// SIMATIC S7-200 project (STEP 7-Micro/WIN), CPU 221 REL 01.10

SYMBOL_TABLE USER1
run              Q0.0
dir              Q0.1
s1               M5.0
s2               M5.1
s3               M5.2
p1               I0.0
p2               I0.1
p3               I0.2
END_SYMBOL_TABLE

ORGANIZATION_BLOCK MAIN:OB1
TITLE=PROGRAM COMMENTS
BEGIN
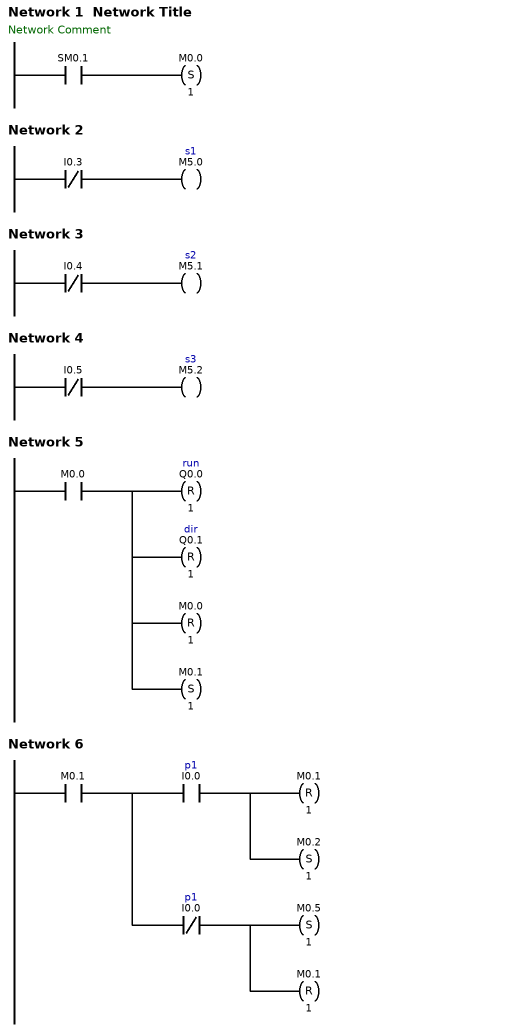
Network 1 // Network Title
// Network Comment
LD     SM0.1
S      M0.0, 1
Network 2
LDN    I0.3
=      s1:M5.0
Network 3
LDN    I0.4
=      s2:M5.1
Network 4
LDN    I0.5
=      s3:M5.2
Network 5
LD     M0.0
R      run:Q0.0, 1
R      dir:Q0.1, 1
R      M0.0, 1
S      M0.1, 1
Network 6
LD     M0.1
LPS
A      p1:I0.0
R      M0.1, 1
S      M0.2, 1
LPP
AN     p1:I0.0
S      M0.5, 1
R      M0.1, 1
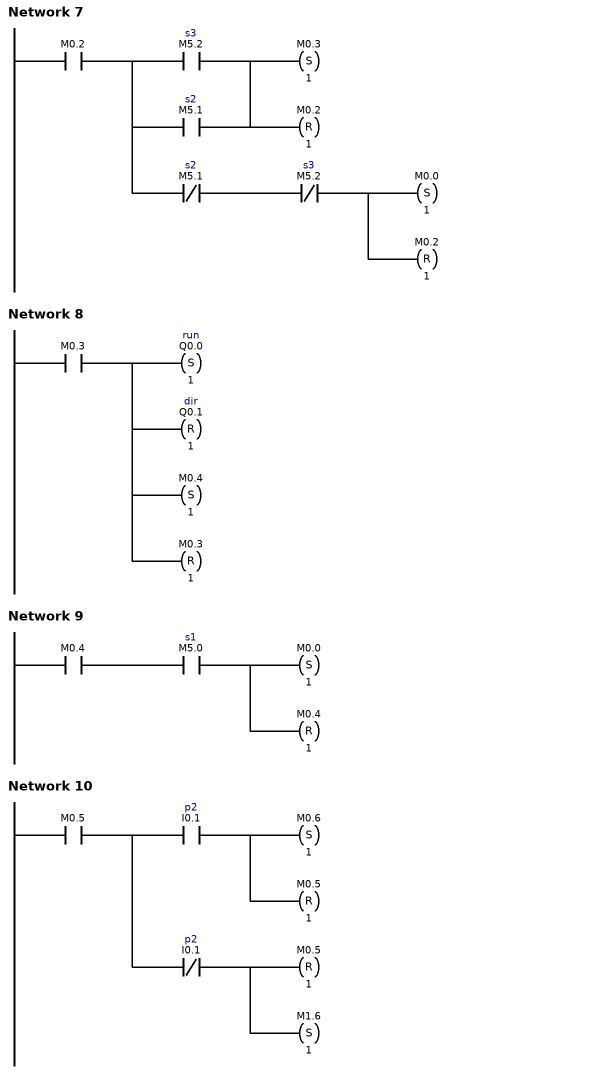
Network 7
LD     M0.2
LPS
LD     s3:M5.2
O      s2:M5.1
ALD
S      M0.3, 1
R      M0.2, 1
LPP
AN     s2:M5.1
AN     s3:M5.2
S      M0.0, 1
R      M0.2, 1
Network 8
LD     M0.3
S      run:Q0.0, 1
R      dir:Q0.1, 1
S      M0.4, 1
R      M0.3, 1
Network 9
LD     M0.4
A      s1:M5.0
S      M0.0, 1
R      M0.4, 1
Network 10
LD     M0.5
LPS
A      p2:I0.1
S      M0.6, 1
R      M0.5, 1
LPP
AN     p2:I0.1
R      M0.5, 1
S      M1.6, 1
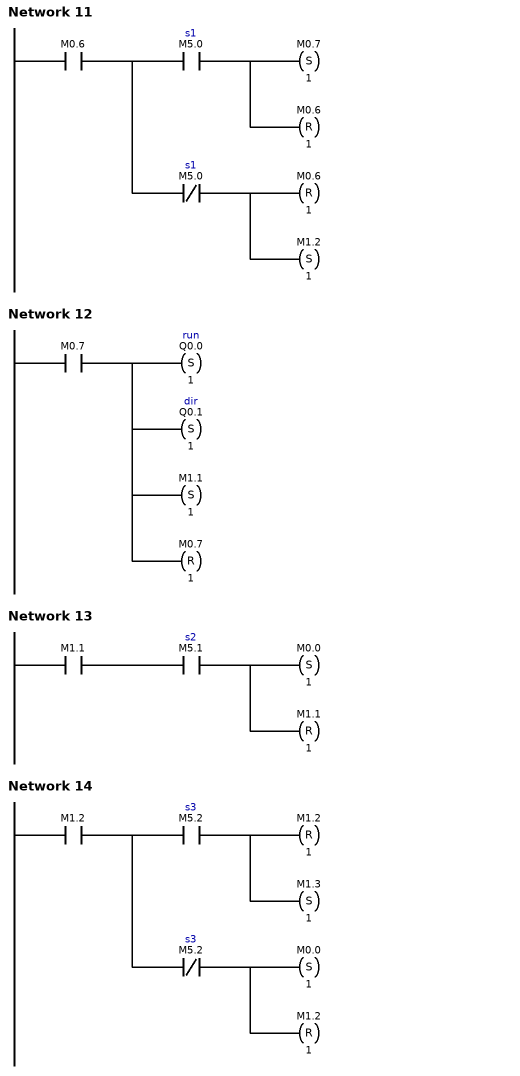
Network 11
LD     M0.6
LPS
A      s1:M5.0
S      M0.7, 1
R      M0.6, 1
LPP
AN     s1:M5.0
R      M0.6, 1
S      M1.2, 1
Network 12
LD     M0.7
S      run:Q0.0, 1
S      dir:Q0.1, 1
S      M1.1, 1
R      M0.7, 1
Network 13
LD     M1.1
A      s2:M5.1
S      M0.0, 1
R      M1.1, 1
Network 14
LD     M1.2
LPS
A      s3:M5.2
R      M1.2, 1
S      M1.3, 1
LPP
AN     s3:M5.2
S      M0.0, 1
R      M1.2, 1
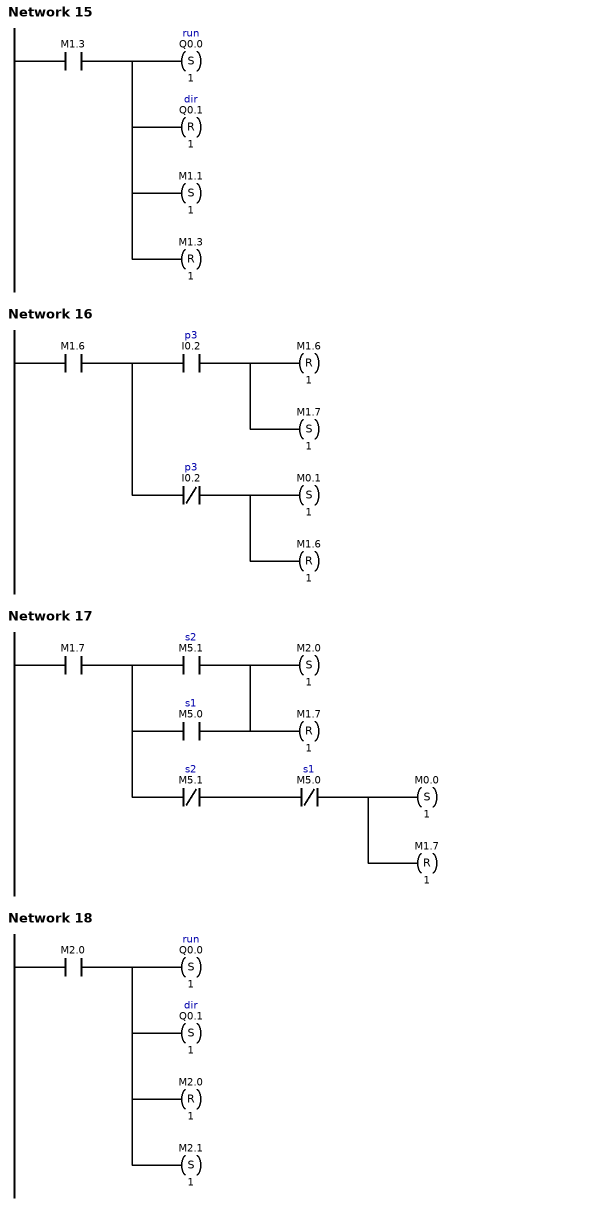
Network 15
LD     M1.3
S      run:Q0.0, 1
R      dir:Q0.1, 1
S      M1.1, 1
R      M1.3, 1
Network 16
LD     M1.6
LPS
A      p3:I0.2
R      M1.6, 1
S      M1.7, 1
LPP
AN     p3:I0.2
S      M0.1, 1
R      M1.6, 1
Network 17
LD     M1.7
LPS
LD     s2:M5.1
O      s1:M5.0
ALD
S      M2.0, 1
R      M1.7, 1
LPP
AN     s2:M5.1
AN     s1:M5.0
S      M0.0, 1
R      M1.7, 1
Network 18
LD     M2.0
S      run:Q0.0, 1
S      dir:Q0.1, 1
R      M2.0, 1
S      M2.1, 1
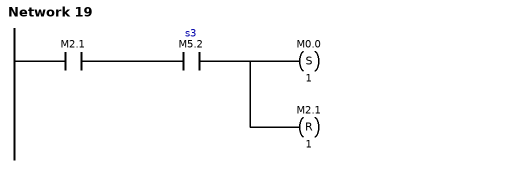
Network 19
LD     M2.1
A      s3:M5.2
S      M0.0, 1
R      M2.1, 1
END_ORGANIZATION_BLOCK
